PROGRAM main
VAR
	Start_Sequence AT %IX0.0 : bool;
	Motor_1 AT %QX0.0 : bool;
	Motor_2 AT %QX0.1 : bool;
	Motor2_Enable : bool;
	TON0 : TON;
END_VAR

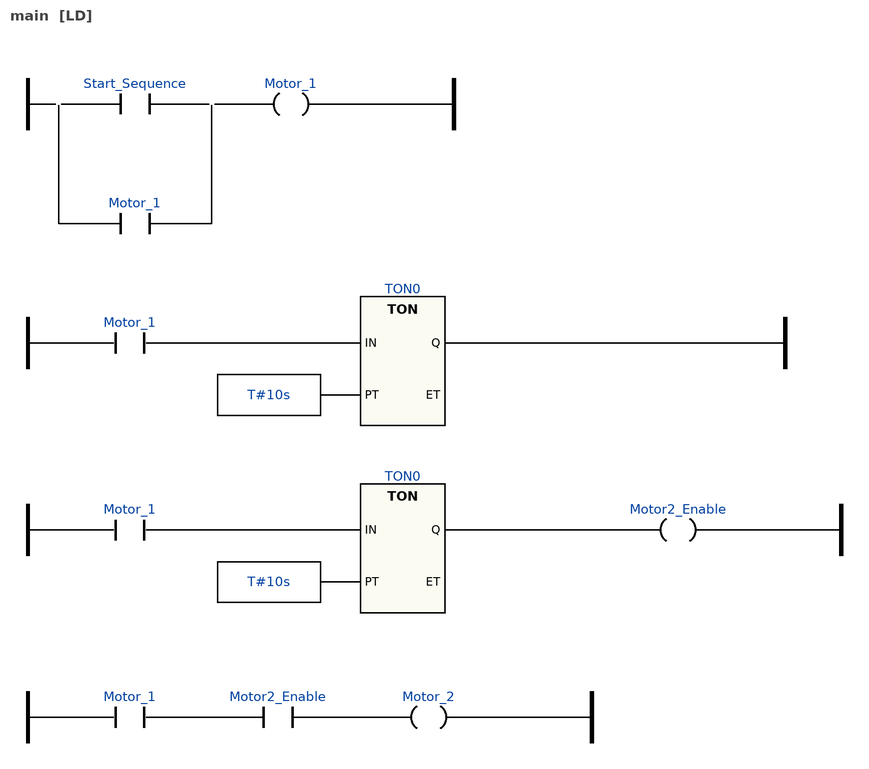
(* LD diagram, written out as Structured Text *)
Motor_1 := Start_Sequence OR Motor_1;
TON0(IN := Motor_1, PT := T#10s);
Motor2_Enable := TON0.Q;
Motor_2 := Motor_1 AND Motor2_Enable;
TON0(IN := Motor_1, PT := T#10s);
END_PROGRAM
